{attribute addProperty BoxType "EL6002-0000-0019"}
{attribute addProperty Id "WcStateAT %I*BIT10.1250InputToggleAT %I*BIT10.1250"}
{attribute addProperty CRC "2560941941"}
{attribute addProperty SizeInBites "2"}
{attribute addProperty SizeInBytes "0.25"}
TYPE WcState_98A4DF75 :
STRUCT
	{attribute addProperty Name "WcState"}
	WcState AT %I* : BOOL;
	{attribute addProperty Name "InputToggle"}
	InputToggle AT %I* : BOOL;
END_STRUCT
END_TYPE

(* stored: Version 1.2.0.0, ProductVersion 3.1.4024.9
   DUT WcState_98A4DF75: Id {fd728343-144b-0980-056f-be61c9668e19} *)
